// TwinCAT 3 PLC project FirstRun_PLC
// ProgramVersion: 3.1.4026.16
// libraries:
//   Tc2_Standard, * (Beckhoff Automation GmbH)
//   Tc2_System, * (Beckhoff Automation GmbH)
// project tree:
//   GVLs/ E_BatteryState.TcDUT
//   / PlcTask.TcTTO
//   POUs/ MAIN.TcPOU
// real-time tasks:
//   TASK PlcTask: cycle T#10ms, priority 20, ADS port 350

CONFIGURATION FirstRun_PLC
    RESOURCE PLC ON TwinCAT3
        TASK PlcTask(INTERVAL := T#10ms, PRIORITY := 20);
        PROGRAM MAIN WITH PlcTask : MAIN;
    END_RESOURCE
END_CONFIGURATION

// ---- GVLs/E_BatteryState.TcDUT
{attribute 'qualified_only'}
{attribute 'strict'}
{attribute 'to_string'}
TYPE E_BatteryState :
(
	Active 			:= 0,
	Gray			:= 1,
	Fault			:= 2,
	Yellow			:= 3
	
);
END_TYPE

// ---- POUs/MAIN.TcPOU
PROGRAM MAIN
VAR
	StartTimer : BOOL;         // Trigger to start the timer
    Timer    : TON;          // TON = On-delay timer
    Output     : BOOL;         // Output after timer elapses

	cycleTime: TIME := T#3S;
	bEllipse: BOOL; 
	
	tCycle: TON;
	cycleTime2: TIME := T#2000MS;
	imageIndex : UINT := 0;   // Index for StateImage
	
	state		: E_BatteryState;
END_VAR

// Trigger the timer
Timer(IN := StartTimer, PT := cycleTime);  // 5-second delay

// Set output when timer is done
Output := Timer.Q;


// Timer logic
tCycle(IN := TRUE, PT := cycleTime2);

IF tCycle.Q THEN
    IF imageIndex < 4 THEN
        imageIndex := imageIndex + 1;
    ELSE
        imageIndex := 0;
    END_IF;

    tCycle(IN := FALSE); // Reset timer
END_IF;

END_PROGRAM
